// TIA Portal V18 export
TYPE "Component Check_ShW"
// stored: IsFailsafeCompliant false
   STRUCT
      Trigger : Bool;
      Q_ID { S7_SetPoint := 'True'} : "ComponentID_ShW";
      IDResult : Int;
      IDResult1 : Array[1..10] of Int;
      Completed : Bool;
   END_STRUCT;
END_TYPE
